// TIA Portal V21 export
// export: Created 2000-01-01T00:00:00.0000000Z, ExportSetting WithDefaults
TagTable "默认变量表"
  HMI_Start : Bool  (PLC tag I_Start, HMI_Connection_1, 100 ms)
  HMI_Stop : Bool  (PLC tag I_Stop, HMI_Connection_1, 100 ms)
  HMI_Run : Bool  (PLC tag Q_Run, HMI_Connection_1, 100 ms)
